    {attribute 'pytmc' := 'pv: IM5L0:PPM:MMS'}
    {attribute 'TcLinkTo' := '.bLimitForwardEnable  := TIIB[IM5L0-EL1084-E4]^Channel 3^Input;
                              .bLimitBackwardEnable := TIIB[IM5L0-EL1084-E4]^Channel 4^Input;
                              .bBrakeRelease        := TIIB[IM5L0-EL2004-E3]^Channel 1^Output;
                              .nRawEncoderULINT     := TIIB[IM5L0-EL5042-E2]^FB Inputs Channel 1^Position'}
    M57: ST_MotionStage := (sName := 'IM5L0:PPM:MMS');

    {attribute 'pytmc' := 'pv: AL1L0:REF:MMS'}
    {attribute 'TcLinkTo' := '.nRawEncoderULINT     := TIIB[AL1L0-EL5042-E2]^FB Inputs Channel 2^Position'}
    M58: ST_MotionStage := (sName := 'AL1L0:REF:MMS');

     // SL2L0-SCATTER: 4 Axes
    {attribute 'pytmc' := 'pv: SL3L0:SCATTER:MMS:BOTTOM'}
    {attribute 'TcLinkTo' := '.bLimitForwardEnable  := TIIB[SL3L0-EL7037-E6]^STM Status^Status^Digital input 1;
                              .bLimitBackwardEnable := TIIB[SL3L0-EL7037-E6]^STM Status^Status^Digital input 2;
                              .nRawEncoderULINT     := TIIB[SL3L0-EL5042-E5]^FB Inputs Channel 1^Position'}
    M59: ST_MotionStage := (sName := 'SL3L0:SCATTER:MMS:BOTTOM');
        {attribute 'pytmc' := 'pv: SL3L0:SCATTER:MMS:TOP'}
    {attribute 'TcLinkTo' := '.bLimitForwardEnable  := TIIB[SL3L0-EL7037-E4]^STM Status^Status^Digital input 1;
                              .bLimitBackwardEnable := TIIB[SL3L0-EL7037-E4]^STM Status^Status^Digital input 2;
                               .nRawEncoderULINT     := TIIB[SL3L0-EL5042-E5]^FB Inputs Channel 2^Position'}
    M60: ST_MotionStage := (sName := 'SL3L0:SCATTER:MMS:TOP');
        {attribute 'pytmc' := 'pv: SL3L0:SCATTER:MMS:SOUTH'}
    {attribute 'TcLinkTo' := '.bLimitForwardEnable  := TIIB[SL3L0-EL7037-E3]^STM Status^Status^Digital input 1;
                              .bLimitBackwardEnable := TIIB[SL3L0-EL7037-E3]^STM Status^Status^Digital input 2;
                                .nRawEncoderULINT     := TIIB[SL3L0-EL5042-E2]^FB Inputs Channel 1^Position'}
    M61: ST_MotionStage := (sName := 'SL3L0:SCATTER:MMS:SOUTH');
    {attribute 'pytmc' := 'pv: SL3L0:SCATTER:MMS:NORTH'}
    {attribute 'TcLinkTo' := '.bLimitForwardEnable  := TIIB[SL3L0-EL7037-E1]^STM Status^Status^Digital input 1;
                              .bLimitBackwardEnable := TIIB[SL3L0-EL7037-E1]^STM Status^Status^Digital input 2;
                            .nRawEncoderULINT     := TIIB[SL3L0-EL5042-E2]^FB Inputs Channel 2^Position'}
    M62: ST_MotionStage := (sName := 'SL3L0:SCATTER:MMS:NORTH');


END_VAR

// ---- Version/Global_Version.TcGVL
{attribute 'TcGenerated'}
{attribute 'no-analysis'}
{attribute 'linkalways'}
// This function has been automatically generated from the project information.
VAR_GLOBAL CONSTANT
	{attribute 'const_non_replaced'}
	stLibVersion_lcls_plc_lfe_motion : ST_LibVersion := (iMajor := 0, iMinor := 0, iBuild := 0, iRevision := 0, nFlags := 0, sVersion := '0.0.0');
END_VAR

// ---- POUs/PRG_1_PlcTask.TcPOU
PROGRAM PRG_1_PlcTask
(*
    Launch site for each component's program
    Only "fast" programs are allowed here,
    anything else needs to be relegated to a second task
*)

PRG_2_PMPS_PRE();

PRG_AT2L0_SOLID();
PRG_IM1L0_XTES();
PRG_IM1L1_PPM();
PRG_IM2L0_XTES();
PRG_IM3L0_PPM();
PRG_IM4L0_XTES();
PRG_IM5L0_PPM();
PRG_PF1L0_WFS();
PRG_RTDSL0();
PRG_SL1L0_POWER();
PRG_SL2L0_POWER();
//PRG_SP1L0_KMONO();
PRG_EM3L0_IPM();
PRG_AL1L0_REF();
PRG_SL3L0_SCATTER();

PRG_3_PMPS_POST();
PRG_4_LOG();

END_PROGRAM

// ---- POUs/PRG_AT2L0_SOLID.TcPOU
PROGRAM PRG_AT2L0_SOLID
VAR
    bAT2L0_debug: BOOL := FALSE;
    nAT2L0_enableMode: ENUM_StageEnableMode := ENUM_StageEnableMode.DURING_MOTION;

    iIndex: INT;
    fbAT2L0_motion: ARRAY [1..19] OF FB_MotionStage;
    fbAT2L0_axes: ARRAY [1..19] OF POINTER TO DUT_MotionStage;
    fbAT2L0_ffo: ARRAY[1..19] OF FB_AttFFO;

    {attribute 'pytmc' := '
        pv: AT2L0:XTES:MMS
        expand: :%.2d:FILTER
    '}
    fbAT2L0_filters: ARRAY[1..19] OF DUT_SATT_Filter;

    {attribute 'pytmc' := '
        pv: AT2L0:XTES:TRANSMISSION
        field: DESC Overall transmission of AT2L0
    '}
    fTransmission: LREAL;

    {attribute 'pytmc' := '
        pv: AT2L0:XTES:MMS
        expand: :%.2d
    '}
    fbAT2L0_states: ARRAY[1..19] OF FB_PositionState1D_InOut;

    stOut: ST_PositionState  := (
        fPosition := 24,
        fDelta := 2,
        fVelocity := 6,
        bMoveOk := TRUE,
        bValid := TRUE);

    stIn: ST_PositionState  := (
        fPosition := 0,
        fDelta := 2,
        fVelocity := 6,
        bMoveOk := TRUE,
        bValid := TRUE);

    // For plotting voltage/current during debugging
    nM1CoilARaw AT %I*: UINT;
    nM1CoilBRaw AT %I*: UINT; // ..CoilBRaw is currently linked to EL7041 'Coil Voltage A'
    nM1CoilA: INT;
    nM1CoilB: INT;
    //nM1Current: INT;
    nM2CoilARaw AT %I*: UINT;
    nM2CoilBRaw AT %I*: UINT;
    nM2CoilA: INT;
    nM2CoilB: INT;
    //nM2Current: INT;
    nM3CoilARaw AT %I*: UINT;
    nM3CoilBRaw AT %I*: UINT;
    nM3CoilA: INT;
    nM3CoilB: INT;
    //nM3Current: INT;
    nM4CoilARaw AT %I*: UINT;
    nM4CoilBRaw AT %I*: UINT;
    nM4CoilA: INT;
    nM4CoilB: INT;
    //nM4Current: INT;
    nM5CoilARaw AT %I*: UINT;
    nM5CoilBRaw AT %I*: UINT;
    nM5CoilA: INT;
    nM5CoilB: INT;
    //nM5Current: INT;
    nM6CoilARaw AT %I*: UINT;
    nM6CoilBRaw AT %I*: UINT;
    nM6CoilA: INT;
    nM6CoilB: INT;
    //nM6Current: INT;
    nM7CoilARaw AT %I*: UINT;
    nM7CoilBRaw AT %I*: UINT;
    nM7CoilA: INT;
    nM7CoilB: INT;
    //nM7Current: INT;
    nM8CoilARaw AT %I*: UINT;
    nM8CoilBRaw AT %I*: UINT;
    nM8CoilA: INT;
    nM8CoilB: INT;
    //nM8Current: INT;
    nM9CoilARaw AT %I*: UINT;
    nM9CoilBRaw AT %I*: UINT;
    nM9CoilA: INT;
    nM9CoilB: INT;
    //nM9Current: INT;
    nM10CoilARaw AT %I*: UINT;
    nM10CoilBRaw AT %I*: UINT;
    nM10CoilA: INT;
    nM10CoilB: INT;
    //nM10Current: INT;
    nM11CoilARaw AT %I*: UINT;
    nM11CoilBRaw AT %I*: UINT;
    nM11CoilA: INT;
    nM11CoilB: INT;
    //nM11Current: INT;
    nM12CoilARaw AT %I*: UINT;
    nM12CoilBRaw AT %I*: UINT;
    nM12CoilA: INT;
    nM12CoilB: INT;
    //nM12Current: INT;
    nM13CoilARaw AT %I*: UINT;
    nM13CoilBRaw AT %I*: UINT;
    nM13CoilA: INT;
    nM13CoilB: INT;
    //nM13Current: INT;
    nM14CoilARaw AT %I*: UINT;
    nM14CoilBRaw AT %I*: UINT;
    nM14CoilA: INT;
    nM14CoilB: INT;
    //nM14Current: INT;
    nM15CoilARaw AT %I*: UINT;
    nM15CoilBRaw AT %I*: UINT;
    nM15CoilA: INT;
    nM15CoilB: INT;
    //nM15Current: INT;
    nM16CoilARaw AT %I*: UINT;
    nM16CoilBRaw AT %I*: UINT;
    nM16CoilA: INT;
    nM16CoilB: INT;
    //nM16Current: INT;
    nM17CoilARaw AT %I*: UINT;
    nM17CoilBRaw AT %I*: UINT;
    nM17CoilA: INT;
    nM17CoilB: INT;
    //nM17Current: INT;
    nM18CoilARaw AT %I*: UINT;
    nM18CoilBRaw AT %I*: UINT;
    nM18CoilA: INT;
    nM18CoilB: INT;
    //nM18Current: INT;
    nM19CoilARaw AT %I*: UINT;
    nM19CoilBRaw AT %I*: UINT;
    nM19CoilA: INT;
    nM19CoilB: INT;
    //nM19Current: INT;

    stFilter : REFERENCE TO DUT_SATT_Filter;
    fFilterDensity : LREAL;
    fFilterAtomicMass : LREAL;
    fbAtomicMass : FB_AtomicMass;
    fbAttenuatorElementDensity : FB_AttenuatorElementDensity;
    fAbsorptionConstant : LREAL;
    bError : BOOL;

END_VAR


fbAT2L0_axes[1]:= ADR(Main.M1);
fbAT2L0_axes[2]:= ADR(Main.M2);
fbAT2L0_axes[3]:= ADR(Main.M3);
fbAT2L0_axes[4]:= ADR(Main.M4);
fbAT2L0_axes[5]:= ADR(Main.M5);
fbAT2L0_axes[6]:= ADR(Main.M6);
fbAT2L0_axes[7]:= ADR(Main.M7);
fbAT2L0_axes[8]:= ADR(Main.M8);
fbAT2L0_axes[9]:= ADR(Main.M9);
fbAT2L0_axes[10]:= ADR(Main.M10);
fbAT2L0_axes[11]:= ADR(Main.M11);
fbAT2L0_axes[12]:= ADR(Main.M12);
fbAT2L0_axes[13]:= ADR(Main.M13);
fbAT2L0_axes[14]:= ADR(Main.M14);
fbAT2L0_axes[15]:= ADR(Main.M15);
fbAT2L0_axes[16]:= ADR(Main.M16);
fbAT2L0_axes[17]:= ADR(Main.M17);
fbAT2L0_axes[18]:= ADR(Main.M18);
fbAT2L0_axes[19]:= ADR(Main.M19);

(* Not a filter *)
fbAT2L0_filters[ 1].fFilterThickness_um := 0;
fbAT2L0_filters[ 1].sFilterMaterial     := '';

fbAT2L0_filters[ 2].fFilterThickness_um := 1280.0;
fbAT2L0_filters[ 2].sFilterMaterial     := 'C';
fbAT2L0_filters[ 3].fFilterThickness_um := 320.0;
fbAT2L0_filters[ 3].sFilterMaterial     := 'C';
fbAT2L0_filters[ 4].fFilterThickness_um := 640.0;
fbAT2L0_filters[ 4].sFilterMaterial     := 'C';
fbAT2L0_filters[ 5].fFilterThickness_um := 160.0;
fbAT2L0_filters[ 5].sFilterMaterial     := 'C';
fbAT2L0_filters[ 6].fFilterThickness_um := 80.0;
fbAT2L0_filters[ 6].sFilterMaterial     := 'C';
fbAT2L0_filters[ 7].fFilterThickness_um := 40.0;
fbAT2L0_filters[ 7].sFilterMaterial     := 'C';
fbAT2L0_filters[ 8].fFilterThickness_um := 20.0;
fbAT2L0_filters[ 8].sFilterMaterial     := 'C';
fbAT2L0_filters[ 9].fFilterThickness_um := 10.0;
fbAT2L0_filters[ 9].sFilterMaterial     := 'C';

fbAT2L0_filters[10].fFilterThickness_um := 10240.0;
fbAT2L0_filters[10].sFilterMaterial     := 'Si';
fbAT2L0_filters[11].fFilterThickness_um := 5120.0;
fbAT2L0_filters[11].sFilterMaterial     := 'Si';
fbAT2L0_filters[12].fFilterThickness_um := 2560.0;
fbAT2L0_filters[12].sFilterMaterial     := 'Si';
fbAT2L0_filters[13].fFilterThickness_um := 1280.0;
fbAT2L0_filters[13].sFilterMaterial     := 'Si';
fbAT2L0_filters[14].fFilterThickness_um := 640.0;
fbAT2L0_filters[14].sFilterMaterial     := 'Si';
fbAT2L0_filters[15].fFilterThickness_um := 320.0;
fbAT2L0_filters[15].sFilterMaterial     := 'Si';
fbAT2L0_filters[16].fFilterThickness_um := 160.0;
fbAT2L0_filters[16].sFilterMaterial     := 'Si';
fbAT2L0_filters[17].fFilterThickness_um := 80.0;
fbAT2L0_filters[17].sFilterMaterial     := 'Si';
fbAT2L0_filters[18].fFilterThickness_um := 40.0;
fbAT2L0_filters[18].sFilterMaterial     := 'Si';
fbAT2L0_filters[19].fFilterThickness_um := 20.0;
fbAT2L0_filters[19].sFilterMaterial     := 'Si';

IF bAT2L0_debug THEN
    nAT2L0_enableMode := ENUM_StageEnableMode.ALWAYS;
ELSE
    nAT2L0_enableMode := ENUM_StageEnableMode.DURING_MOTION;
END_IF


(* Recalculate the overall transmission below *)
fTransmission := 1.0;

FOR iIndex := 1 TO 19 DO
    fbAT2L0_motion[iIndex](stMotionStage := fbAT2L0_axes[iIndex]^);
    fbAT2L0_axes[iIndex]^.nEnableMode := nAT2L0_enableMode;
    fbAT2L0_axes[iIndex]^.bHardwareEnable := TRUE;
    fbAT2L0_axes[iIndex]^.bPowerSelf := TRUE;
    stFilter REF= fbAT2L0_filters[iIndex];

    fbAT2L0_states[iIndex](
        stMotionStage := fbAT2L0_axes[iIndex]^,
        stOut := stOut,
        stIn := stIn);

    fbAT2L0_ffo[iIndex](
        stMotionStage := fbAT2L0_axes[iIndex]^,
        enumState := fbAT2L0_states[iIndex].eStateGet,
        fbFFHWO := GVL.fbFastFaultOutput1);

    IF fbAT2L0_states[iIndex].eStateGet = ENUM_EpicsInOut.UNKNOWN THEN
        stFilter.fTransmission := 0.0;
    ELSIF fbAT2L0_states[iIndex].eStateGet = ENUM_EpicsInOut.OUT OR stFilter.sFilterMaterial = '' THEN
        stFilter.fTransmission := 1.0;
    ELSE
        fbAtomicMass(sName:=stFilter.sFilterMaterial, fValue=>fFilterAtomicMass);
        fbAttenuatorElementDensity(sName:=stFilter.sFilterMaterial, fDensity=>fFilterDensity);

        fAbsorptionConstant := F_CalculateAbsorptionConstant(
            sElement:=stFilter.sFilterMaterial,
            fEnergyEV:=PMPS_GVL.stCurrentBeamParameters.neV,
            fDensity_gm3:=fFilterDensity,
            fAtomicWeight:=fFilterAtomicMass,
            bError=>bError,
        );
        stFilter.fTransmission := F_CalculateTransmission(
            fAbsorptionConstant:=fAbsorptionConstant,
            fThickness_in_m:=stFilter.fFilterThickness_um * 1.0E-6
        );
    END_IF

    fTransmission := fTransmission * stFilter.fTransmission;
END_FOR

IF fbAT2L0_states[1].eStateGet = ENUM_EpicsInOut.IN THEN
    (* Inspection mirror blocks the beam *)
    GVL.rCurTrans[PMPS.L_Attenuators.AT2L0].nTran := 0.0;
    (* TODO fast fault as well *)
ELSE
    GVL.rCurTrans[PMPS.L_Attenuators.AT2L0].nTran := LREAL_TO_REAL(fTransmission);
END_IF

iIndex := 0;

nM1CoilA := UINT_TO_INT(nM1CoilARaw);
nM1CoilB := UINT_TO_INT(nM1CoilBRaw);
//nM1Current := ABS(nM1CoilA) + ABS(nM1CoilB);
nM2CoilA := UINT_TO_INT(nM2CoilARaw);
nM2CoilB := UINT_TO_INT(nM2CoilBRaw);
//nM2Current := ABS(nM2CoilA) + ABS(nM2CoilB);
nM3CoilA := UINT_TO_INT(nM3CoilARaw);
nM3CoilB := UINT_TO_INT(nM3CoilBRaw);
//nM3Current := ABS(nM3CoilA) + ABS(nM3CoilB);
nM4CoilA := UINT_TO_INT(nM4CoilARaw);
nM4CoilB := UINT_TO_INT(nM4CoilBRaw);
//nM4Current := ABS(nM4CoilA) + ABS(nM4CoilB);
nM5CoilA := UINT_TO_INT(nM5CoilARaw);
nM5CoilB := UINT_TO_INT(nM5CoilBRaw);
//nM5Current := ABS(nM5CoilA) + ABS(nM5CoilB);
nM5CoilA := UINT_TO_INT(nM5CoilARaw);
nM5CoilB := UINT_TO_INT(nM5CoilBRaw);
//nM5Current := ABS(nM5CoilA) + ABS(nM5CoilB);
nM6CoilA := UINT_TO_INT(nM6CoilARaw);
nM6CoilB := UINT_TO_INT(nM6CoilBRaw);
//nM6Current := ABS(nM6CoilA) + ABS(nM6CoilB);
nM7CoilA := UINT_TO_INT(nM7CoilARaw);
nM7CoilB := UINT_TO_INT(nM7CoilBRaw);
//nM7Current := ABS(nM7CoilA) + ABS(nM7CoilB);
nM8CoilA := UINT_TO_INT(nM8CoilARaw);
nM8CoilB := UINT_TO_INT(nM8CoilBRaw);
//nM8Current := ABS(nM9CoilA) + ABS(nM9CoilB);
nM9CoilA := UINT_TO_INT(nM9CoilARaw);
nM9CoilB := UINT_TO_INT(nM9CoilBRaw);
//nM9Current := ABS(nM9CoilA) + ABS(nM9CoilB);
nM10CoilA := UINT_TO_INT(nM10CoilARaw);
nM10CoilB := UINT_TO_INT(nM10CoilBRaw);
//nM10Current := ABS(nM10CoilA) + ABS(nM10CoilB);
nM11CoilA := UINT_TO_INT(nM11CoilARaw);
nM11CoilB := UINT_TO_INT(nM11CoilBRaw);
//nM11Current := ABS(nM11CoilA) + ABS(nM11CoilB);
nM12CoilA := UINT_TO_INT(nM12CoilARaw);
nM12CoilB := UINT_TO_INT(nM12CoilBRaw);
//nM12Current := ABS(nM12CoilA) + ABS(nM12CoilB);
nM13CoilA := UINT_TO_INT(nM13CoilARaw);
nM13CoilB := UINT_TO_INT(nM13CoilBRaw);
//nM13Current := ABS(nM13CoilA) + ABS(nM13CoilB);
nM14CoilA := UINT_TO_INT(nM14CoilARaw);
nM14CoilB := UINT_TO_INT(nM14CoilBRaw);
//nM14Current := ABS(nM14CoilA) + ABS(nM14CoilB);
nM15CoilA := UINT_TO_INT(nM15CoilARaw);
nM15CoilB := UINT_TO_INT(nM15CoilBRaw);
//nM15Current := ABS(nM15CoilA) + ABS(nM15CoilB);
nM16CoilA := UINT_TO_INT(nM16CoilARaw);
nM16CoilB := UINT_TO_INT(nM16CoilBRaw);
//nM16Current := ABS(nM16CoilA) + ABS(nM16CoilB);
nM17CoilA := UINT_TO_INT(nM17CoilARaw);
nM17CoilB := UINT_TO_INT(nM17CoilBRaw);
//nM17Current := ABS(nM17CoilA) + ABS(nM17CoilB);
nM18CoilA := UINT_TO_INT(nM18CoilARaw);
nM18CoilB := UINT_TO_INT(nM18CoilBRaw);
//nM18Current := ABS(nM2CoilA) + ABS(nM18CoilB);
nM19CoilA := UINT_TO_INT(nM19CoilARaw);
nM19CoilB := UINT_TO_INT(nM19CoilBRaw);
//nM19Current := ABS(nM2CoilA) + ABS(nM2CoilB);

END_PROGRAM

// ---- POUs/PRG_IM1L0_XTES.TcPOU
PROGRAM PRG_IM1L0_XTES
VAR
    {attribute 'pytmc' := '
        pv: IM1L0:XTES
        io: io
    '}
    {attribute 'TcLinkTo' := '.bZoomEndFwd := TIIB[IM1L0-EL1088]^Channel 1^Input;
                              .bZoomEndBwd := TIIB[IM1L0-EL1088]^Channel 2^Input;
                              .bFocusEndFwd := TIIB[IM1L0-EL1088]^Channel 3^Input;
                              .bFocusEndBwd := TIIB[IM1L0-EL1088]^Channel 4^Input;
                              .fbOpal.bOpalPower := TIIB[IM1L0-EL2004]^Channel 2^Output;
                              .fbLED.bLedPower := TIIB[IM1L0-EL2004]^Channel 3^Output'}
    fbIM1L0: FB_XPIM;
    {attribute 'pytmc' := '
        pv: IM1L0:XTES:FLOW_OK
        field: ZNAM LOW
        field: ONAM OK
    '}
    {attribute 'TcLinkTo' := 'TIIB[IM1L0-EL7342]^DCM Status Channel 1^Status^Digital input 1'}
    bIM1L0FlowOk AT %I*: BOOL;
    {attribute 'TcLinkTo' := '.Status := TIIB[IM1L0-EL6002]^COM TxPDO-Map Inputs Channel 1^Status;
                              .D[0] := TIIB[IM1L0-EL6002]^COM TxPDO-Map Inputs Channel 1^Data In 0;
                              .D[1] := TIIB[IM1L0-EL6002]^COM TxPDO-Map Inputs Channel 1^Data In 1;
                              .D[2] := TIIB[IM1L0-EL6002]^COM TxPDO-Map Inputs Channel 1^Data In 2;
                              .D[3] := TIIB[IM1L0-EL6002]^COM TxPDO-Map Inputs Channel 1^Data In 3;
                              .D[4] := TIIB[IM1L0-EL6002]^COM TxPDO-Map Inputs Channel 1^Data In 4;
                              .D[5] := TIIB[IM1L0-EL6002]^COM TxPDO-Map Inputs Channel 1^Data In 5;
                              .D[6] := TIIB[IM1L0-EL6002]^COM TxPDO-Map Inputs Channel 1^Data In 6;
                              .D[7] := TIIB[IM1L0-EL6002]^COM TxPDO-Map Inputs Channel 1^Data In 7;
                              .D[8] := TIIB[IM1L0-EL6002]^COM TxPDO-Map Inputs Channel 1^Data In 8;
                              .D[9] := TIIB[IM1L0-EL6002]^COM TxPDO-Map Inputs Channel 1^Data In 9;
                              .D[10] := TIIB[IM1L0-EL6002]^COM TxPDO-Map Inputs Channel 1^Data In 10;
                              .D[11] := TIIB[IM1L0-EL6002]^COM TxPDO-Map Inputs Channel 1^Data In 11;
                              .D[12] := TIIB[IM1L0-EL6002]^COM TxPDO-Map Inputs Channel 1^Data In 12;
                              .D[13] := TIIB[IM1L0-EL6002]^COM TxPDO-Map Inputs Channel 1^Data In 13;
                              .D[14] := TIIB[IM1L0-EL6002]^COM TxPDO-Map Inputs Channel 1^Data In 14;
                              .D[15] := TIIB[IM1L0-EL6002]^COM TxPDO-Map Inputs Channel 1^Data In 15;
                              .D[16] := TIIB[IM1L0-EL6002]^COM TxPDO-Map Inputs Channel 1^Data In 16;
                              .D[17] := TIIB[IM1L0-EL6002]^COM TxPDO-Map Inputs Channel 1^Data In 17;
                              .D[18] := TIIB[IM1L0-EL6002]^COM TxPDO-Map Inputs Channel 1^Data In 18;
                              .D[19] := TIIB[IM1L0-EL6002]^COM TxPDO-Map Inputs Channel 1^Data In 19;
                              .D[20] := TIIB[IM1L0-EL6002]^COM TxPDO-Map Inputs Channel 1^Data In 20;
                              .D[21] := TIIB[IM1L0-EL6002]^COM TxPDO-Map Inputs Channel 1^Data In 21'}
    stEL6In AT %I*: EL6InData22b;
    {attribute 'TcLinkTo' := '.Ctrl := TIIB[IM1L0-EL6002]^COM RxPDO-Map Outputs Channel 1^Ctrl;
                              .D[0] := TIIB[IM1L0-EL6002]^COM RxPDO-Map Outputs Channel 1^Data Out 0;
                              .D[1] := TIIB[IM1L0-EL6002]^COM RxPDO-Map Outputs Channel 1^Data Out 1;
                              .D[2] := TIIB[IM1L0-EL6002]^COM RxPDO-Map Outputs Channel 1^Data Out 2;
                              .D[3] := TIIB[IM1L0-EL6002]^COM RxPDO-Map Outputs Channel 1^Data Out 3;
                              .D[4] := TIIB[IM1L0-EL6002]^COM RxPDO-Map Outputs Channel 1^Data Out 4;
                              .D[5] := TIIB[IM1L0-EL6002]^COM RxPDO-Map Outputs Channel 1^Data Out 5;
                              .D[6] := TIIB[IM1L0-EL6002]^COM RxPDO-Map Outputs Channel 1^Data Out 6;
                              .D[7] := TIIB[IM1L0-EL6002]^COM RxPDO-Map Outputs Channel 1^Data Out 7;
                              .D[8] := TIIB[IM1L0-EL6002]^COM RxPDO-Map Outputs Channel 1^Data Out 8;
                              .D[9] := TIIB[IM1L0-EL6002]^COM RxPDO-Map Outputs Channel 1^Data Out 9;
                              .D[10] := TIIB[IM1L0-EL6002]^COM RxPDO-Map Outputs Channel 1^Data Out 10;
                              .D[11] := TIIB[IM1L0-EL6002]^COM RxPDO-Map Outputs Channel 1^Data Out 11;
                              .D[12] := TIIB[IM1L0-EL6002]^COM RxPDO-Map Outputs Channel 1^Data Out 12;
                              .D[13] := TIIB[IM1L0-EL6002]^COM RxPDO-Map Outputs Channel 1^Data Out 13;
                              .D[14] := TIIB[IM1L0-EL6002]^COM RxPDO-Map Outputs Channel 1^Data Out 14;
                              .D[15] := TIIB[IM1L0-EL6002]^COM RxPDO-Map Outputs Channel 1^Data Out 15;
                              .D[16] := TIIB[IM1L0-EL6002]^COM RxPDO-Map Outputs Channel 1^Data Out 16;
                              .D[17] := TIIB[IM1L0-EL6002]^COM RxPDO-Map Outputs Channel 1^Data Out 17;
                              .D[18] := TIIB[IM1L0-EL6002]^COM RxPDO-Map Outputs Channel 1^Data Out 18;
                              .D[19] := TIIB[IM1L0-EL6002]^COM RxPDO-Map Outputs Channel 1^Data Out 19;
                              .D[20] := TIIB[IM1L0-EL6002]^COM RxPDO-Map Outputs Channel 1^Data Out 20;
                              .D[21] := TIIB[IM1L0-EL6002]^COM RxPDO-Map Outputs Channel 1^Data Out 21'}
    stEL6Out AT %Q*: EL6OutData22b;

    fbStateSetup: FB_StateSetupHelper;
    stDefault: ST_PositionState := (
        fVelocity := 1,
        bMoveOk := TRUE,
        bValid := TRUE
    );
END_VAR


fbStateSetup(stPositionState:=stDefault, bSetDefault:=TRUE);
fbStateSetup(stPositionState:=fbIM1L0.stOut, fPosition:=0,          sPmpsState:='IM1L0:XTES-OUT');
fbStateSetup(stPositionState:=fbIM1L0.stYag, fPosition:=-86.65,     sPmpsState:='IM1L0:XTES-YAG');
fbStateSetup(stPositionState:=fbIM1L0.stDiamond, fPosition:=-56.65, sPmpsState:='IM1L0:XTES-DIAMOND');
fbStateSetup(stPositionState:=fbIM1L0.stReticle, fPosition:=-26.65, sPmpsState:='IM1L0:XTES-RETICLE');

fbIM1L0(
    fbArbiter := GVL.fbArbiter,
    fbFFHWO := GVL.fbFastFaultOutput1a,
    stYStage := Main.M20,
    stZoomStage := Main.M21,
    stFocusStage := Main.M22,
    stEl6In := stEL6In,
    stEl6Out := stEl6Out,
    sDeviceName := 'IM1L0:XTES',
    sTransitionKey := 'IM1L0:XTES-TRANSITION',
    bEnableMotion := TRUE,
    bEnableBeamParams := TRUE,
    bEnablePositionLimits := TRUE,
);

END_PROGRAM

// ---- POUs/PRG_IM2L0_XTES.TcPOU
PROGRAM PRG_IM2L0_XTES
VAR
    {attribute 'pytmc' := '
        pv: IM2L0:XTES
        io: io
    '}
    {attribute 'TcLinkTo' := '.bZoomEndFwd := TIIB[IM2L0-EL1088]^Channel 1^Input;
                              .bZoomEndBwd := TIIB[IM2L0-EL1088]^Channel 2^Input;
                              .bFocusEndFwd := TIIB[IM2L0-EL1088]^Channel 3^Input;
                              .bFocusEndBwd := TIIB[IM2L0-EL1088]^Channel 4^Input;
                              .fbOpal.bOpalPower := TIIB[IM2L0-EL2004]^Channel 2^Output;
                              .fbLED.bLedPower := TIIB[IM2L0-EL2004]^Channel 3^Output'}
    fbIM2L0: FB_XPIM;
    {attribute 'TcLinkTo' := '.Status := TIIB[IM2L0-EL6002]^COM TxPDO-Map Inputs Channel 1^Status;
                              .D[0] := TIIB[IM2L0-EL6002]^COM TxPDO-Map Inputs Channel 1^Data In 0;
                              .D[1] := TIIB[IM2L0-EL6002]^COM TxPDO-Map Inputs Channel 1^Data In 1;
                              .D[2] := TIIB[IM2L0-EL6002]^COM TxPDO-Map Inputs Channel 1^Data In 2;
                              .D[3] := TIIB[IM2L0-EL6002]^COM TxPDO-Map Inputs Channel 1^Data In 3;
                              .D[4] := TIIB[IM2L0-EL6002]^COM TxPDO-Map Inputs Channel 1^Data In 4;
                              .D[5] := TIIB[IM2L0-EL6002]^COM TxPDO-Map Inputs Channel 1^Data In 5;
                              .D[6] := TIIB[IM2L0-EL6002]^COM TxPDO-Map Inputs Channel 1^Data In 6;
                              .D[7] := TIIB[IM2L0-EL6002]^COM TxPDO-Map Inputs Channel 1^Data In 7;
                              .D[8] := TIIB[IM2L0-EL6002]^COM TxPDO-Map Inputs Channel 1^Data In 8;
                              .D[9] := TIIB[IM2L0-EL6002]^COM TxPDO-Map Inputs Channel 1^Data In 9;
                              .D[10] := TIIB[IM2L0-EL6002]^COM TxPDO-Map Inputs Channel 1^Data In 10;
                              .D[11] := TIIB[IM2L0-EL6002]^COM TxPDO-Map Inputs Channel 1^Data In 11;
                              .D[12] := TIIB[IM2L0-EL6002]^COM TxPDO-Map Inputs Channel 1^Data In 12;
                              .D[13] := TIIB[IM2L0-EL6002]^COM TxPDO-Map Inputs Channel 1^Data In 13;
                              .D[14] := TIIB[IM2L0-EL6002]^COM TxPDO-Map Inputs Channel 1^Data In 14;
                              .D[15] := TIIB[IM2L0-EL6002]^COM TxPDO-Map Inputs Channel 1^Data In 15;
                              .D[16] := TIIB[IM2L0-EL6002]^COM TxPDO-Map Inputs Channel 1^Data In 16;
                              .D[17] := TIIB[IM2L0-EL6002]^COM TxPDO-Map Inputs Channel 1^Data In 17;
                              .D[18] := TIIB[IM2L0-EL6002]^COM TxPDO-Map Inputs Channel 1^Data In 18;
                              .D[19] := TIIB[IM2L0-EL6002]^COM TxPDO-Map Inputs Channel 1^Data In 19;
                              .D[20] := TIIB[IM2L0-EL6002]^COM TxPDO-Map Inputs Channel 1^Data In 20;
                              .D[21] := TIIB[IM2L0-EL6002]^COM TxPDO-Map Inputs Channel 1^Data In 21'}
    stEL6In AT %I*: EL6InData22b;
    {attribute 'TcLinkTo' := '.Ctrl := TIIB[IM2L0-EL6002]^COM RxPDO-Map Outputs Channel 1^Ctrl;
                              .D[0] := TIIB[IM2L0-EL6002]^COM RxPDO-Map Outputs Channel 1^Data Out 0;
                              .D[1] := TIIB[IM2L0-EL6002]^COM RxPDO-Map Outputs Channel 1^Data Out 1;
                              .D[2] := TIIB[IM2L0-EL6002]^COM RxPDO-Map Outputs Channel 1^Data Out 2;
                              .D[3] := TIIB[IM2L0-EL6002]^COM RxPDO-Map Outputs Channel 1^Data Out 3;
                              .D[4] := TIIB[IM2L0-EL6002]^COM RxPDO-Map Outputs Channel 1^Data Out 4;
                              .D[5] := TIIB[IM2L0-EL6002]^COM RxPDO-Map Outputs Channel 1^Data Out 5;
                              .D[6] := TIIB[IM2L0-EL6002]^COM RxPDO-Map Outputs Channel 1^Data Out 6;
                              .D[7] := TIIB[IM2L0-EL6002]^COM RxPDO-Map Outputs Channel 1^Data Out 7;
                              .D[8] := TIIB[IM2L0-EL6002]^COM RxPDO-Map Outputs Channel 1^Data Out 8;
                              .D[9] := TIIB[IM2L0-EL6002]^COM RxPDO-Map Outputs Channel 1^Data Out 9;
                              .D[10] := TIIB[IM2L0-EL6002]^COM RxPDO-Map Outputs Channel 1^Data Out 10;
                              .D[11] := TIIB[IM2L0-EL6002]^COM RxPDO-Map Outputs Channel 1^Data Out 11;
                              .D[12] := TIIB[IM2L0-EL6002]^COM RxPDO-Map Outputs Channel 1^Data Out 12;
                              .D[13] := TIIB[IM2L0-EL6002]^COM RxPDO-Map Outputs Channel 1^Data Out 13;
                              .D[14] := TIIB[IM2L0-EL6002]^COM RxPDO-Map Outputs Channel 1^Data Out 14;
                              .D[15] := TIIB[IM2L0-EL6002]^COM RxPDO-Map Outputs Channel 1^Data Out 15;
                              .D[16] := TIIB[IM2L0-EL6002]^COM RxPDO-Map Outputs Channel 1^Data Out 16;
                              .D[17] := TIIB[IM2L0-EL6002]^COM RxPDO-Map Outputs Channel 1^Data Out 17;
                              .D[18] := TIIB[IM2L0-EL6002]^COM RxPDO-Map Outputs Channel 1^Data Out 18;
                              .D[19] := TIIB[IM2L0-EL6002]^COM RxPDO-Map Outputs Channel 1^Data Out 19;
                              .D[20] := TIIB[IM2L0-EL6002]^COM RxPDO-Map Outputs Channel 1^Data Out 20;
                              .D[21] := TIIB[IM2L0-EL6002]^COM RxPDO-Map Outputs Channel 1^Data Out 21'}
    stEL6Out AT %Q*: EL6OutData22b;

    fbStateSetup: FB_StateSetupHelper;
    stDefault: ST_PositionState := (
        fVelocity := 1,
        bMoveOk := TRUE,
        bValid := TRUE
    );

    {attribute 'TcLinkTo' := 'TIIB[IM2L0-EL7041]^STM Status^Status^Digital input 1'}
    bDefectiveLimitSwitch AT %I*: BOOL;
END_VAR


fbStateSetup(stPositionState:=stDefault, bSetDefault:=TRUE);
fbStateSetup(stPositionState:=fbIM2L0.stOut, fPosition:=0,          sPmpsState:='IM2L0:XTES-OUT');
fbStateSetup(stPositionState:=fbIM2L0.stYag, fPosition:=-87.65,     sPmpsState:='IM2L0:XTES-YAG');
fbStateSetup(stPositionState:=fbIM2L0.stDiamond, fPosition:=-57.65, sPmpsState:='IM2L0:XTES-DIAMOND');
fbStateSetup(stPositionState:=fbIM2L0.stReticle, fPosition:=-27.65, sPmpsState:='IM2L0:XTES-RETICLE');

Main.M24.bLimitForwardEnable := bDefectiveLimitSwitch OR (Main.M24.stAxisStatus.fActPosition < 0);

fbIM2L0(
    fbArbiter := GVL.fbArbiter,
    fbFFHWO := GVL.fbFastFaultOutput1a,
    stYStage := Main.M24,
    stZoomStage := Main.M25,
    stFocusStage := Main.M26,
    stEl6In := stEL6In,
    stEl6Out := stEl6Out,
    sDeviceName := 'IM2L0:XTES',
    sTransitionKey := 'IM2L0:XTES-TRANSITION',
    bEnableMotion := TRUE,
    bEnableBeamParams := TRUE,
    bEnablePositionLimits := TRUE,
);

END_PROGRAM

// ---- POUs/PRG_IM3L0_PPM.TcPOU
PROGRAM PRG_IM3L0_PPM
VAR
    {attribute 'pytmc' := '
        pv: IM3L0:PPM
        io: io
    '}
    {attribute 'TcLinkTo' := '.fbGige.iIlluminatorINT := TIIB[IM3L0-EL4004]^AO Outputs Channel 1^Analog output;
                              .fbGige.bGigePower := TIIB[IM3L0-EL2004]^Channel 2^Output;
                              .fbPowerMeter.iVoltageINT := TIIB[IM3L0-EL3062]^AI Standard Channel 1^Value;
                              .fbPowerMeter.fbTempSensor.bError := TIIB[IM3L0-EL3314]^TC Inputs Channel 1^Status^Error;
                              .fbPowerMeter.fbTempSensor.bUnderrange := TIIB[IM3L0-EL3314]^TC Inputs Channel 1^Status^Underrange;
                              .fbPowerMeter.fbTempSensor.bOverrange := TIIB[IM3L0-EL3314]^TC Inputs Channel 1^Status^Overrange;
                              .fbPowerMeter.fbTempSensor.iRaw := TIIB[IM3L0-EL3314]^TC Inputs Channel 1^Value;
                              .fbYagTempSensor.bError := TIIB[IM3L0-EL3314]^TC Inputs Channel 2^Status^Error;
                              .fbYagTempSensor.bUnderrange := TIIB[IM3L0-EL3314]^TC Inputs Channel 2^Status^Underrange;
                              .fbYagTempSensor.bOverrange := TIIB[IM3L0-EL3314]^TC Inputs Channel 2^Status^Overrange;
                              .fbYagTempSensor.iRaw := TIIB[IM3L0-EL3314]^TC Inputs Channel 2^Value'}
    fbIM3L0: FB_PPM;

    fbStateSetup: FB_StateSetupHelper;
    stDefault: ST_PositionState := (
        fVelocity := 10,
        bMoveOk := TRUE,
        bValid := TRUE
    );
END_VAR


fbStateSetup(stPositionState:=stDefault, bSetDefault:=TRUE);
fbStateSetup(stPositionState:=fbIM3L0.stOut, fPosition:=-8.40,    sPmpsState:='IM3L0:PPM-OUT');
fbStateSetup(stPositionState:=fbIM3L0.stPower, fPosition:=-47.40, sPmpsState:='IM3L0:PPM-POWERMETER');
fbStateSetup(stPositionState:=fbIM3L0.stYag1, fPosition:=-71.50,  sPmpsState:='IM3L0:PPM-YAG1');
fbStateSetup(stPositionState:=fbIM3L0.stYag2, fPosition:=-97.51,  sPmpsState:='IM3L0:PPM-YAG2');

fbIM3L0(
    fbArbiter := GVL.fbArbiter,
    fbFFHWO := GVL.fbFastFaultOutput1c,
    stYStage := Main.M27,
    sDeviceName := 'IM3L0:PPM',
    sTransitionKey := 'IM3L0:PPM-TRANSITION',
    bEnableMotion := TRUE,
    bEnableBeamParams := TRUE,
    bEnablePositionLimits := TRUE,
    fResponsivity := 0.0506,
);

END_PROGRAM

// ---- POUs/PRG_IM4L0_XTES.TcPOU
PROGRAM PRG_IM4L0_XTES
VAR
    {attribute 'pytmc' := '
        pv: IM4L0:XTES
        io: io
    '}
    {attribute 'TcLinkTo' := '.bZoomEndFwd := TIIB[IM4L0-EL1088]^Channel 1^Input;
                              .bZoomEndBwd := TIIB[IM4L0-EL1088]^Channel 2^Input;
                              .bFocusEndFwd := TIIB[IM4L0-EL1088]^Channel 3^Input;
                              .bFocusEndBwd := TIIB[IM4L0-EL1088]^Channel 4^Input;
                              .fbOpal.bOpalPower := TIIB[IM4L0-EL2004]^Channel 2^Output;
                              .fbLED.bLedPower := TIIB[IM4L0-EL2004]^Channel 3^Output'}
    fbIM4L0: FB_XPIM;
    {attribute 'TcLinkTo' := '.Status := TIIB[IM4L0-EL6002]^COM TxPDO-Map Inputs Channel 1^Status;
                              .D[0] := TIIB[IM4L0-EL6002]^COM TxPDO-Map Inputs Channel 1^Data In 0;
                              .D[1] := TIIB[IM4L0-EL6002]^COM TxPDO-Map Inputs Channel 1^Data In 1;
                              .D[2] := TIIB[IM4L0-EL6002]^COM TxPDO-Map Inputs Channel 1^Data In 2;
                              .D[3] := TIIB[IM4L0-EL6002]^COM TxPDO-Map Inputs Channel 1^Data In 3;
                              .D[4] := TIIB[IM4L0-EL6002]^COM TxPDO-Map Inputs Channel 1^Data In 4;
                              .D[5] := TIIB[IM4L0-EL6002]^COM TxPDO-Map Inputs Channel 1^Data In 5;
                              .D[6] := TIIB[IM4L0-EL6002]^COM TxPDO-Map Inputs Channel 1^Data In 6;
                              .D[7] := TIIB[IM4L0-EL6002]^COM TxPDO-Map Inputs Channel 1^Data In 7;
                              .D[8] := TIIB[IM4L0-EL6002]^COM TxPDO-Map Inputs Channel 1^Data In 8;
                              .D[9] := TIIB[IM4L0-EL6002]^COM TxPDO-Map Inputs Channel 1^Data In 9;
                              .D[10] := TIIB[IM4L0-EL6002]^COM TxPDO-Map Inputs Channel 1^Data In 10;
                              .D[11] := TIIB[IM4L0-EL6002]^COM TxPDO-Map Inputs Channel 1^Data In 11;
                              .D[12] := TIIB[IM4L0-EL6002]^COM TxPDO-Map Inputs Channel 1^Data In 12;
                              .D[13] := TIIB[IM4L0-EL6002]^COM TxPDO-Map Inputs Channel 1^Data In 13;
                              .D[14] := TIIB[IM4L0-EL6002]^COM TxPDO-Map Inputs Channel 1^Data In 14;
                              .D[15] := TIIB[IM4L0-EL6002]^COM TxPDO-Map Inputs Channel 1^Data In 15;
                              .D[16] := TIIB[IM4L0-EL6002]^COM TxPDO-Map Inputs Channel 1^Data In 16;
                              .D[17] := TIIB[IM4L0-EL6002]^COM TxPDO-Map Inputs Channel 1^Data In 17;
                              .D[18] := TIIB[IM4L0-EL6002]^COM TxPDO-Map Inputs Channel 1^Data In 18;
                              .D[19] := TIIB[IM4L0-EL6002]^COM TxPDO-Map Inputs Channel 1^Data In 19;
                              .D[20] := TIIB[IM4L0-EL6002]^COM TxPDO-Map Inputs Channel 1^Data In 20;
                              .D[21] := TIIB[IM4L0-EL6002]^COM TxPDO-Map Inputs Channel 1^Data In 21'}
    stEL6In AT %I*: EL6InData22b;
    {attribute 'TcLinkTo' := '.Ctrl := TIIB[IM4L0-EL6002]^COM RxPDO-Map Outputs Channel 1^Ctrl;
                              .D[0] := TIIB[IM4L0-EL6002]^COM RxPDO-Map Outputs Channel 1^Data Out 0;
                              .D[1] := TIIB[IM4L0-EL6002]^COM RxPDO-Map Outputs Channel 1^Data Out 1;
                              .D[2] := TIIB[IM4L0-EL6002]^COM RxPDO-Map Outputs Channel 1^Data Out 2;
                              .D[3] := TIIB[IM4L0-EL6002]^COM RxPDO-Map Outputs Channel 1^Data Out 3;
                              .D[4] := TIIB[IM4L0-EL6002]^COM RxPDO-Map Outputs Channel 1^Data Out 4;
                              .D[5] := TIIB[IM4L0-EL6002]^COM RxPDO-Map Outputs Channel 1^Data Out 5;
                              .D[6] := TIIB[IM4L0-EL6002]^COM RxPDO-Map Outputs Channel 1^Data Out 6;
                              .D[7] := TIIB[IM4L0-EL6002]^COM RxPDO-Map Outputs Channel 1^Data Out 7;
                              .D[8] := TIIB[IM4L0-EL6002]^COM RxPDO-Map Outputs Channel 1^Data Out 8;
                              .D[9] := TIIB[IM4L0-EL6002]^COM RxPDO-Map Outputs Channel 1^Data Out 9;
                              .D[10] := TIIB[IM4L0-EL6002]^COM RxPDO-Map Outputs Channel 1^Data Out 10;
                              .D[11] := TIIB[IM4L0-EL6002]^COM RxPDO-Map Outputs Channel 1^Data Out 11;
                              .D[12] := TIIB[IM4L0-EL6002]^COM RxPDO-Map Outputs Channel 1^Data Out 12;
                              .D[13] := TIIB[IM4L0-EL6002]^COM RxPDO-Map Outputs Channel 1^Data Out 13;
                              .D[14] := TIIB[IM4L0-EL6002]^COM RxPDO-Map Outputs Channel 1^Data Out 14;
                              .D[15] := TIIB[IM4L0-EL6002]^COM RxPDO-Map Outputs Channel 1^Data Out 15;
                              .D[16] := TIIB[IM4L0-EL6002]^COM RxPDO-Map Outputs Channel 1^Data Out 16;
                              .D[17] := TIIB[IM4L0-EL6002]^COM RxPDO-Map Outputs Channel 1^Data Out 17;
                              .D[18] := TIIB[IM4L0-EL6002]^COM RxPDO-Map Outputs Channel 1^Data Out 18;
                              .D[19] := TIIB[IM4L0-EL6002]^COM RxPDO-Map Outputs Channel 1^Data Out 19;
                              .D[20] := TIIB[IM4L0-EL6002]^COM RxPDO-Map Outputs Channel 1^Data Out 20;
                              .D[21] := TIIB[IM4L0-EL6002]^COM RxPDO-Map Outputs Channel 1^Data Out 21'}
    stEL6Out AT %Q*: EL6OutData22b;

     {attribute 'pytmc' := 'pv: IM4L0:SCRP:LED:01:PWR
                        io: io
                        field: ZNAM OFF
                        field: ONAM ON
     '}

     {attribute 'TcLinkTo' := 'TIIB[IM4L0-EL2004]^Channel 4^Output'}
    bIM4L0_SCRP_LED_01 AT %Q*: BOOL;

    fbStateSetup: FB_StateSetupHelper;
    stDefault: ST_PositionState := (
        fVelocity := 1,
        bMoveOk := TRUE,
        bValid := TRUE
    );
END_VAR


fbStateSetup(stPositionState:=stDefault, bSetDefault:=TRUE);
fbStateSetup(stPositionState:=fbIM4L0.stOut, fPosition:=0,          sPmpsState:='IM4L0:XTES-OUT');
fbStateSetup(stPositionState:=fbIM4L0.stYag, fPosition:=-86.65,     sPmpsState:='IM4L0:XTES-YAG');
fbStateSetup(stPositionState:=fbIM4L0.stDiamond, fPosition:=-56.65, sPmpsState:='IM4L0:XTES-DIAMOND');
fbStateSetup(stPositionState:=fbIM4L0.stReticle, fPosition:=-26.65, sPmpsState:='IM4L0:XTES-RETICLE');

fbIM4L0(
    fbArbiter := GVL.fbArbiter,
    fbFFHWO := GVL.fbFastFaultOutput1b,
    stYStage := Main.M28,
    stZoomStage := Main.M29,
    stFocusStage := Main.M30,
    stEl6In := stEL6In,
    stEl6Out := stEl6Out,
    sDeviceName := 'IM4L0:XTES',
    sTransitionKey := 'IM4L0:XTES-TRANSITION',
    bEnableMotion := TRUE,
    bEnableBeamParams := TRUE,
    bEnablePositionLimits := TRUE,
);

END_PROGRAM

// ---- POUs/PRG_IM5L0_PPM.TcPOU
PROGRAM PRG_IM5L0_PPM
VAR
    {attribute 'pytmc' := '
        pv: IM5L0:PPM
        io: io
    '}
    {attribute 'TcLinkTo' := '.fbGige.iIlluminatorINT := TIIB[IM5L0-EL4004-E7]^AO Outputs Channel 1^Analog output;
                              .fbPowerMeter.iVoltageINT := TIIB[IM5L0-EL3602-E6]^AI Inputs Channel 1^Value;
                              .fbPowerMeter.fbTempSensor.bError := TIIB[IM5L0-EL3202-0010-E5]^RTD Inputs Channel 1^Status^Error;
                              .fbPowerMeter.fbTempSensor.bUnderrange := TIIB[IM5L0-EL3202-0010-E5]^RTD Inputs Channel 1^Status^Underrange;
                              .fbPowerMeter.fbTempSensor.bOverrange := TIIB[IM5L0-EL3202-0010-E5]^RTD Inputs Channel 1^Status^Overrange;
                              .fbPowerMeter.fbTempSensor.iRaw := TIIB[IM5L0-EL3202-0010-E5]^RTD Inputs Channel 1^Value'}
    fbIM5L0: FB_PPM;

    fbStateSetup: FB_StateSetupHelper;
    stDefault: ST_PositionState := (
        fVelocity := 0.5,
        bMoveOk := TRUE,
        bValid := TRUE
    );
END_VAR

//'fbIM5L0.fbPowerMeter.fbTempSensor.fResolution :=0.01;

fbStateSetup(stPositionState:=stDefault, bSetDefault:=TRUE);
fbStateSetup(stPositionState:=fbIM5L0.stOut, fPosition:=-3.0004, 	sPmpsState:='IM5L0:PPM-OUT');
fbStateSetup(stPositionState:=fbIM5L0.stPower, fPosition:=-43.3451, sPmpsState:='IM5L0:PPM-POWERMETER');
fbStateSetup(stPositionState:=fbIM5L0.stYag1, fPosition:=-65.39670,	sPmpsState:='IM5L0:PPM-YAG1');
fbStateSetup(stPositionState:=fbIM5L0.stYag2, fPosition:=-76.0395, 	sPmpsState:='IM5L0:PPM-YAG2');

fbIM5L0(
    fbArbiter := GVL.fbArbiter,
    fbFFHWO := GVL.fbFastFaultOutput1d,
    stYStage := Main.M57,
    sDeviceName := 'IM5L0:PPM',
    sTransitionKey := 'IM5L0:PPM-TRANSITION',
    bEnableMotion := TRUE,
    bEnableBeamParams := TRUE,
    bEnablePositionLimits := TRUE,
    fResponsivity := 1.0,
    iTermBits := 31,
    fTermMax := 10000,
    fTermMin := -10000
);

END_PROGRAM

// ---- POUs/PRG_PF1L0_WFS.TcPOU
PROGRAM PRG_PF1L0_WFS
VAR
    {attribute 'pytmc' := '
        pv: PF1L0:WFS
        io: io
    '}
    {attribute 'TcLinkTo' := '.fbThermoCouple1.bError := TIIB[PF1L0-EL3314]^TC Inputs Channel 1^Status^Error;
                              .fbThermoCouple1.bUnderrange := TIIB[PF1L0-EL3314]^TC Inputs Channel 1^Status^Underrange;
                              .fbThermoCouple1.bOverrange := TIIB[PF1L0-EL3314]^TC Inputs Channel 1^Status^Overrange;
                              .fbThermoCouple1.iRaw := TIIB[PF1L0-EL3314]^TC Inputs Channel 1^Value;
                              .fbThermoCouple2.bError := TIIB[PF1L0-EL3314]^TC Inputs Channel 2^Status^Error;
                              .fbThermoCouple2.bUnderrange := TIIB[PF1L0-EL3314]^TC Inputs Channel 2^Status^Underrange;
                              .fbThermoCouple2.bOverrange := TIIB[PF1L0-EL3314]^TC Inputs Channel 2^Status^Overrange;
                              .fbThermoCouple2.iRaw := TIIB[PF1L0-EL3314]^TC Inputs Channel 2^Value'}
    fbPF1L0: FB_WFS;
    stSiBP: ST_BeamParams := PMPS_GVL.cstFullBeam;
    stFoilBP: ST_BeamParams := PMPS_GVL.cstFullBeam;

    fbStateSetup: FB_StateSetupHelper;
    stDefault: ST_PositionState := (
        fVelocity := 1,
        bMoveOk := TRUE,
        bValid := TRUE
    );
END_VAR


fbStateSetup(stPositionState:=stDefault, bSetDefault:=TRUE);
fbStateSetup(stPositionState:=fbPF1L0.stOut, fPosition:=-13,         sPmpsState:='PF1L0:WFS-OUT');
fbStateSetup(stPositionState:=fbPF1L0.stTarget1, fPosition:=-93.77,  sPmpsState:='PF1L0:WFS-TARGET1');
fbStateSetup(stPositionState:=fbPF1L0.stTarget2, fPosition:=-79.402, sPmpsState:='PF1L0:WFS-TARGET2');
fbStateSetup(stPositionState:=fbPF1L0.stTarget3, fPosition:=-65.028, sPmpsState:='PF1L0:WFS-TARGET3');
fbStateSetup(stPositionState:=fbPF1L0.stTarget4, fPosition:=-50.652, sPmpsState:='PF1L0:WFS-TARGET4');
fbStateSetup(stPositionState:=fbPF1L0.stTarget5, fPosition:=-36.277, sPmpsState:='PF1L0:WFS-TARGET5');

fbPF1L0(
    fbArbiter := GVL.fbArbiter,
    fbFFHWO := GVL.fbFastFaultOutput1b,
    stYStage := Main.M31,
    stZStage := Main.M32,
    sDeviceName := 'PF1L0:WFS',
    sTransitionKey := 'PF1L0:WFS-TRANSITION',
    bEnableMotion := TRUE,
    bEnableBeamParams := TRUE,
    bEnablePositionLimits := TRUE,
    eEnumGet => GVL.ePF1L0State,
);

END_PROGRAM

// ---- POUs/PRG_EM3L0_IPM.TcPOU
PROGRAM PRG_EM3L0_IPM
VAR
    {attribute 'pytmc' := '
        pv: EM3L0:IPM
        io: io
    '}
    fbEM3L0: FB_IPM;

    fbStateSetup: FB_StateSetupHelper;
    stDefault: ST_PositionState :=(
        fVelocity := 0.5,
        bMoveOK := TRUE,
        bValid := TRUE
    );
END_VAR


fbStateSetup(StPositionState:=stDefault, bSetDefault:=TRUE);
fbStateSetup(StPositionState:=fbEM3L0.stOut, fposition:=0, sPmpsState := 'EM3L0:IPM-OUT');
fbStateSetup(StPositionState:=fbEM3L0.stTarget1, fposition:=-18, sPmpsState := 'EM3L0:IPM-TARGET1');
fbStateSetup(StPositionState:=fbEM3L0.stTarget2, fposition:=-38.6, sPmpsState := 'EM3L0:IPM-TARGET2');
fbStateSetup(StPositionState:=fbEM3L0.stTarget3, fposition:=-59.15, sPmpsState := 'EM3L0:IPM-TARGET3');
fbStateSetup(StPositionState:=fbEM3L0.stTarget4, fposition:=-79.85, sPmpsState := 'EM3L0:IPM-TARGET4');

fbEM3L0(
    fbArbiter := GVL.fbArbiter,
    fbFFHWO := GVL.fbFastFaultOutput1c,
    stXStage := MAIN.M55,
    stYStage := MAIN.M56,
    sDeviceName := 'EM3L0:IPM',
    sTransitionKey := 'EM3L0:IPM-TRANSITION',
    bEnableMotion := TRUE,
    bEnableBeamParams := TRUE,
    bEnablePositionLimits := TRUE
);

END_PROGRAM

// ---- POUs/PRG_AL1L0_REF.TcPOU
PROGRAM PRG_AL1L0_REF
VAR
    {attribute 'pytmc' := 'pv: AL1L0:REF'}
    {attribute 'TcLinkTo' := '.fbLaser.iLaserINT := TIIB[AL1L0-EL4004-E4]^AO Outputs Channel 1^Analog output;
                              .fbLaser.iShutdownINT := TIIB[AL1L0-EL4004-E4]^AO Outputs Channel 2^Analog output'}
    fbAL1L0: FB_REF;

    fbStateSetup: FB_StateSetupHelper;
    stDefault: ST_PositionState := (
        fVelocity := 1,
        bMoveOk := TRUE,
        bValid := TRUE
    );
END_VAR

//Device doesn't have end of travel limits switches
MAIN.M58.bLimitBackwardEnable := TRUE;
MAIN.M58.bLimitForwardEnable := TRUE;


fbStateSetup(stPositionState:=stDefault, bSetDefault:=TRUE);
fbStateSetup(stPositionState:=fbAL1L0.stOut, fPosition:=0, sPmpsState:='AL1L0:REF-OUT');
fbStateSetup(stPositionState:=fbAL1L0.stIn, fPosition:=-43.38, fDelta:=2, sPmpsState:='AL1L0:REF-IN');

fbAL1L0(
    fbFFHWO := GVL.fbFastFaultOutput1d,
    fbArbiter := GVL.fbArbiter,
    stYStage := MAIN.M58,
    sDeviceName := 'AL1L0:REF',
    sTransitionKey := 'AL1L0:REF-TRANSITION',
    bEnableMotion := TRUE,
    bEnableBeamParams := TRUE,
    bEnablePositionLimits := TRUE,
);

END_PROGRAM

// ---- POUs/PRG_SL3L0_SCATTER.TcPOU
PROGRAM PRG_SL3L0_SCATTER
VAR // linking to rtd in the following order Bottom - South - TOP - NORTH
    {attribute 'pytmc' := '
        pv: SL3L0:SCATTER
        io: io
    '}
    fbSL3L0: FB_SLITS_SCATTER;

    {attribute 'pytmc' := '
    pv: SL3L0:SCATTER:GO;
    io: io;
    field: ZNAM False;
    field: ONAM True;
    '}
    bExecuteMotion:BOOL ;

    bMoveOk:BOOL :=TRUE;

     (*Offsets*)
    (* Absolute encoder value at the HLS + Absolute encoder value at the centered beam *)
    rEncoderOffsetTop: REAL := 20;
    rEncoderOffsetBottom: REAL := -20;
    rEncoderOffsetNorth: REAL := 20;
    rEncoderOffsetSouth: REAL := -20;

END_VAR


(*
--MAPPING TO PHYSICAL TERMINAL--
Main.M59     (Bottom)
Main.M61     (South)
Main.M60     (Top)
Main.M62     (North)
*)
//Absolute enocders
Main.M59.nHomingMode := ENUM_EpicsHomeCmd.NONE;
Main.M60.nHomingMode := ENUM_EpicsHomeCmd.NONE;
Main.M61.nHomingMode := ENUM_EpicsHomeCmd.NONE;
Main.M62.nHomingMode := ENUM_EpicsHomeCmd.NONE;

fbSL3L0.rEncoderOffsetTop := rEncoderOffsetTop;
fbSL3L0.rEncoderOffsetBottom := rEncoderOffsetBottom;
fbSL3L0.rEncoderOffsetNorth := rEncoderOffsetNorth;
fbSL3L0.rEncoderOffsetSouth := rEncoderOffsetSouth;

fbSL3L0.bMoveOk := bMoveOk;
fbSL3L0(stTopBlade:=  Main.M60,
        stBottomBlade:= Main.M59,
        stNorthBlade:=  Main.M62,
        stSouthBlade:=  Main.M61,
        bExecuteMotion:=bExecuteMotion);

END_PROGRAM

// ---- Temp/FB_SLITS_SCATTER.TcPOU
FUNCTION_BLOCK FB_SLITS_SCATTER EXTENDS FB_SLITS
VAR_INPUT
END_VAR
VAR_OUTPUT
END_VAR
VAR
END_VAR

ACT_init();
// Instantiate Function block for all the blades
ACT_Motion();
//SET and GET the requested and Actual values
ACT_CalculatePositions();

END_FUNCTION_BLOCK

// ---- POUs/PRG_3_PMPS_POST.TcPOU
PROGRAM PRG_3_PMPS_POST
VAR
    fbArbiterIO: FB_SubSysToArbiter_IO;
    bMR1L1_Veto_OUT: BOOL;
    fbVetoArbiter_L1: FB_VetoArbiter;
	//Fast Fault to Aggregate all Group 1 faults
	g_FastFault		:	FB_FastFault;
	g_FastFaultOutput2: INT;
	q_xFastFaultOut: INT;
END_VAR

bMR1L1_Veto_OUT := PMPS_GVL.stCurrentBeamParameters.aVetoDevices[PMPS.L_Stopper.MR1L1_OUT] AND NOT PMPS_GVL.stCurrentBeamParameters.aVetoDevices[PMPS.L_Stopper.MR1L1_IN];

GVL.fbFastFaultOutput1.Execute();
GVL.fbFastFaultOutput1a.Execute();
GVL.fbFastFaultOutput2.Execute(i_xVeto:=bMR1L1_Veto_OUT);

// Aggregate FastFaultOutputs into a single FastFault
g_FastFault(
    io_fbFFHWO := GVL.fbFastFaultOutput1,
    i_xOK := (  GVL.fbFastFaultOutput1a.q_xFastFaultOut
                AND GVL.fbFastFaultOutput1b.q_xFastFaultOut
				AND GVL.fbFastFaultOutput1c.q_xFastFaultOut
				AND GVL.fbFastFaultOutput1d.q_xFastFaultOut
             ),
    i_xAutoReset:=TRUE
);




fbVetoArbiter_L1(bVeto:=bMR1L1_Veto_OUT,
                HigherAuthority := GVL.fbArbiter,
                LowerAuthority := GVL.fbArbiter2,
                FFO := GVL.fbFastFaultOutput1);

fbArbiterIO(
    Arbiter:=GVL.fbArbiter,
    fbFFHWO:=GVL.fbFastFaultOutput1);

END_PROGRAM
